{attribute 'GeneratedUsingTerminal: IL2300-B110-0016'}
{attribute addProperty BoxType "IL2300-B110-0016"}
{attribute addProperty Id "Term_19KL_D4CFBC220Term_390_Ix1000KL_8EF4D3E90"}
{attribute addProperty CRC "2895154398"}
{attribute addProperty Size "0"}
TYPE A_0019_IL2300_B110_0016_AC908CDE EXTENDS IL2300_A2FCADE7 :
STRUCT
	{attribute addProperty Name "Term_19"}
	Term_19 : KL_D4CFBC22;
	{attribute addProperty Name "Term_390_Ix1000"}
	Term_390_Ix1000 : KL_8EF4D3E9;
END_STRUCT
END_TYPE

(* stored: Version 1.2.0.0, ProductVersion 3.1.4024.9
   DUT A_0019_IL2300_B110_0016_AC908CDE: Id {8e8e3437-71d8-448e-9dc1-fc144f221746} *)
